INTERFACE I_Pump

PROPERTY ControlMode : E_PumpControlMode
GET
END_GET
SET
END_SET
END_PROPERTY

PROPERTY Error : BOOL
GET
END_GET
SET
END_SET
END_PROPERTY

PROPERTY Info : ST_PumpInfo
GET
END_GET
SET
END_SET
END_PROPERTY

METHOD Run : BOOL
VAR_INPUT
END_VAR
END_METHOD

PROPERTY SetOn : BOOL
GET
END_GET
SET
END_SET
END_PROPERTY

PROPERTY Setpoint : REAL
GET
END_GET
SET
END_SET
END_PROPERTY

END_INTERFACE

(* stored: Version 1.1.0.1, ProductVersion 3.1.4022.10
   Itf I_Pump: Id {6708c869-51bd-40b3-85aa-c589ee8ef940}
   Property ControlMode: Id {0c419dd5-76f6-4e27-b46f-fb91615d6acb}
   Get Get: Id {d3938a8c-818a-4dc4-bd8a-4d69883e8b26}
   Set Set: Id {aacf2ae1-d420-415d-aadd-1f477c6bd076}
   Property Error: Id {dde96706-37f3-487d-8277-4e32acc9a409}
   Get Get: Id {953246e6-062b-4759-815f-3762378fed07}
   Set Set: Id {399a5c66-b7a5-42ea-8095-3c70092fa7d1}
   Property Info: Id {33af2e0f-377e-42f2-9e4d-304d1b2354ce}
   Get Get: Id {3e0b9307-ea45-4500-9648-62f76348eb87}
   Set Set: Id {6d636757-d2a9-4963-91a7-766327cdb211}
   Method Run: Id {a5dd7c0b-b49f-48a9-8ae0-91e8b008cb3c}
   Property SetOn: Id {0e587226-d53a-4505-86c2-9b0e3da39fbf}
   Get Get: Id {29b7ae73-716f-4194-bb7b-ea08bd2b176d}
   Set Set: Id {5a240b5b-4035-478f-ab0b-537a602dfd77}
   Property Setpoint: Id {32eec7ee-8c7c-4301-9b66-d3ba251bbd5e}
   Get Get: Id {7ecb7839-204c-4cec-b5dd-4fd3c3fdb67f}
   Set Set: Id {310b12d6-57d6-4b9d-b739-dc957067b719} *)
